// Mitsubishi GX Works2 project: part 2   PLC: FX3G

// global labels: Global1
VAR_GLOBAL
  start_button AT X001 : BOOL;
  on_light AT Y001 : BOOL;
  on_indication AT M0 : BOOL;
  moist AT X004 : BOOL;
  End_Timer AT TC1 : BOOL;
END_VAR
VAR_GLOBAL CONSTANT
  const_20 : INT := 200;
END_VAR
VAR_GLOBAL
  mixer AT Y002 : BOOL;
  temp_180 AT X003 : BOOL;
  temp_200 AT X002 : BOOL;
  timer_out AT TS1 : BOOL;
  heat AT Y003 : BOOL;
END_VAR

// task Task_01 (event TRUE, interval 0, priority 31): POU_01

PROGRAM POU_01
(* structured ladder/FBD written out as ST: instructions are called as NAME(EN, inputs, outputs); _pN, _eN, _tN stand for wires *)
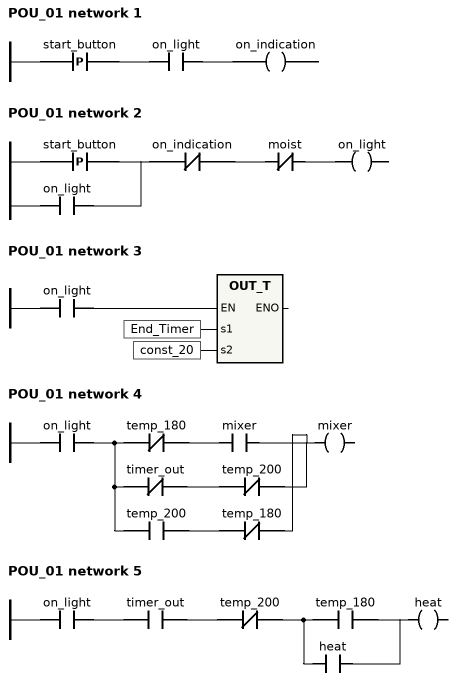
(* network 1 *)
on_indication := LDP(TRUE, start_button) AND on_light;
(* network 2 *)
on_light := ((LDP(TRUE, start_button) OR on_light) AND NOT on_indication) AND NOT moist;
(* network 3 *)
OUT_T(on_light, End_Timer, const_20);
(* network 4 *)
mixer := (on_light AND NOT temp_180 AND mixer) OR (on_light AND NOT timer_out AND NOT temp_200) OR (on_light AND temp_200 AND NOT temp_180);
(* network 5 *)
_p1 := on_light AND timer_out AND NOT temp_200;
heat := (_p1 AND temp_180) OR (_p1 AND heat);
END_PROGRAM
